# EPICS autosave request: dlmApp/Db/dlm_settings.req
$(P)$(Q)sampleCriterion
$(P)$(Q)sampleThreshold
$(P)$(Q)sampleIxLow
$(P)$(Q)sampleIxHigh
$(P)$(Q)histogram
$(P)$(Q)histNumVoltBins
$(P)$(Q)histVoltsLow
$(P)$(Q)histVoltsHigh
file acalcout_settings.req P=$(P)$(Q)acalcDebug
